// TwinCAT 3 PLC project ModbusExt_Sample
// ProgramVersion: 3.1.4026.27
// libraries:
//   ModbusExt2, * (Beckhoff Automation)
//   Tc2_SerialCom, * (Beckhoff Automation GmbH)
//   Tc2_Standard, * (Beckhoff Automation GmbH)
//   Tc2_System, * (Beckhoff Automation GmbH)
//   Tc2_Utilities, * (Beckhoff Automation GmbH)
// project tree:
//   GVLs/ GVL_IO.TcGVL, GVL_Site.TcGVL
//   / PlcTask.TcTTO
//   POUs/ MAIN.TcPOU
//   POUs/Profiles/ FB_Mb_AbbCorMeter.TcPOU, FB_Mb_DiagDemo.TcPOU, FB_Mb_FlowMeter.TcPOU, FB_Mb_TestGood.TcPOU, FB_Mb_TestValve123.TcPOU
// (motion and I/O tree: see PLC project modbusext2)
// real-time tasks:
//   TASK PlcTask1: cycle T#10ms, priority 21, ADS port 351
//   TASK PlcTask: cycle T#10ms, priority 20, ADS port 350

CONFIGURATION ModbusExt_Sample
    RESOURCE PLC ON TwinCAT3
        TASK PlcTask(INTERVAL := T#10ms, PRIORITY := 20);
        PROGRAM MAIN WITH PlcTask : MAIN;
    END_RESOURCE
END_CONFIGURATION

// ---- GVLs/GVL_IO.TcGVL
{attribute 'qualified_only'}
VAR_GLOBAL
	stEl6In1  AT %I* : EL6inData22B;
	stEl6Out1 AT %Q* : EL6outData22B;
END_VAR

// ---- GVLs/GVL_Site.TcGVL
{attribute 'qualified_only'}
VAR_GLOBAL
	{attribute 'TcInitSymbol'}
	sTcpHost   : STRING(15) := '127.0.0.1';
	{attribute 'TcInitSymbol'}
	nTcpPort   : UINT := 502;
	{attribute 'TcInitSymbol'}
	nDemoUnit  : USINT := 1;
	{attribute 'TcInitSymbol'}
	nMeterUnit : USINT := 1;
END_VAR

// ---- POUs/MAIN.TcPOU
PROGRAM MAIN
VAR
	// Transports — call before the devices that use them
	fbTcp          : FB_MbTransportTcp;
	fbRs485        : FB_MbTransportRtu;

	// Devices
	fbDemo         : FB_Mb_DiagDemo;
	fbMeter        : FB_Mb_TestGood;
	fbTemp		   : FB_ModbusDevice;

	// Write handshake example
	fSetpointCmd   : LREAL;
	bWriteSetpoint : BOOL;
END_VAR

// ---- Transports ----
fbTcp(sHost := GVL_Site.sTcpHost, nPort := GVL_Site.nTcpPort);
fbRs485(pComIn := ADR(GVL_IO.stEl6In1), pComOut := ADR(GVL_IO.stEl6Out1), nSizeComIn := SIZEOF(GVL_IO.stEl6In1));

// ---- Devices ----
fbDemo(itfTransport := fbTcp,   nUnitId := GVL_Site.nDemoUnit,  bEnable := TRUE);
fbMeter(itfTransport := fbRs485, nUnitId := GVL_Site.nMeterUnit, bEnable := TRUE, sLogName := 'FlowMeter_Inlet');

// ---- Write handshake: set fSetpointCmd, pulse bWriteSetpoint ----
IF bWriteSetpoint AND NOT fbDemo.Setpoint.bWriteReq AND NOT fbDemo.Setpoint.bWriteBusy THEN
	fbDemo.Setpoint.fWriteValue := fSetpointCmd;
	fbDemo.Setpoint.bWriteReq   := TRUE;
END_IF

IF fbDemo.Setpoint.bWriteDone OR fbDemo.Setpoint.bWriteErr THEN
	fbDemo.Setpoint.bWriteReq := FALSE;
	bWriteSetpoint            := FALSE;
END_IF

END_PROGRAM

// ---- POUs/Profiles/FB_Mb_DiagDemo.TcPOU
(*@ModbusExt.Profile v1 - managed by ModbusExt Profile Editor. One point per line.*)
FUNCTION_BLOCK FB_Mb_DiagDemo EXTENDS FB_ModbusDevice
VAR_INPUT
	Setpoint : ST_MbPoint := (nAddr := 40001);   // UInt16, read and write
	Flow     : ST_MbPoint := (nAddr := 40003, eType := E_MbType.Real32);   // 2 registers
	Temp     : ST_MbPoint := (nAddr := 40005, eType := E_MbType.Int16, fRawMin := 0, fRawMax := 1000, fEngMin := 0, fEngMax := 100, bUseFailValue := TRUE, fFailValue := -1);   // scaled, fails to -1
	Run      : ST_MbPoint := (nAddr := 1);   // coil
	Fault    : ST_MbPoint := (nAddr := 10001, ePoll := E_MbPoll.Slow);   // discrete input, slow
	Amps     : ST_MbPoint := (nAddr := 40007, eType := E_MbType.Int16);   // Test with chad and kyle, lord please work
	Volts	 : ST_MbPoint := (nAddr := 40008, eType := E_MbType.Int16);		// Test manually added from inside TC
END_VAR

Register();
SUPER^();

METHOD Register
Profile(sModel := 'DiagslaveDemo', eWordOrder := E_MbWordOrder.CDAB, tSlowPoll := T#2S);
AddPoint(Setpoint, 'Setpoint');
AddPoint(Flow, 'Flow');
AddPoint(Temp, 'Temp');
AddPoint(Run, 'Run');
AddPoint(Fault, 'Fault');
AddPoint(Amps, 'Amps');
END_METHOD

END_FUNCTION_BLOCK

// ---- POUs/Profiles/FB_Mb_TestGood.TcPOU
FUNCTION_BLOCK FB_Mb_TestGood EXTENDS FB_ModbusDevice
VAR_INPUT
	// Holding registers: 40001..40004 contiguous, 40010 within gap 8 -> one block
	Hr1    : ST_MbPoint := (nAddr := 40001);
	Hr2    : ST_MbPoint := (nAddr := 40002, eType := E_MbType.Int16, fRawMin := 0, fRawMax := 1000, fEngMin := 0, fEngMax := 100);
	Hr3    : ST_MbPoint := (nAddr := 40003, eType := E_MbType.Real32);
	Hr4    : ST_MbPoint := (nAddr := 40010, eType := E_MbType.UInt32);
	// Gap > 8 -> second block
	Hr5    : ST_MbPoint := (nAddr := 40100, eType := E_MbType.Text, nRegs := 8);
	// Slow -> its own block
	Hr6    : ST_MbPoint := (nAddr := 40116, ePoll := E_MbPoll.Slow);
	// Off -> no block
	Hr7    : ST_MbPoint := (nAddr := 40200, ePoll := E_MbPoll.Off);
	// Far away -> third fast HR block
	Hr8    : ST_MbPoint := (nAddr := 40400);
	Hr9    : ST_MbPoint := (nAddr := 40410);
	Hr10   : ST_MbPoint := (nAddr := 40420);
	Status : ST_MbPoint := (nAddr := 40300, eType := E_MbType.RegisterBit, nBit := 3);
	// Input registers, contiguous -> one block
	Ir1    : ST_MbPoint := (nAddr := 30001, eType := E_MbType.Real32);
	Ir2    : ST_MbPoint := (nAddr := 30003, eType := E_MbType.UInt32);
	// Coils and a discrete input
	Coil1  : ST_MbPoint := (nAddr := 1);
	Coil2  : ST_MbPoint := (nAddr := 2);
	Di1    : ST_MbPoint := (nAddr := 10001);
END_VAR

Register();
SUPER^();

//FB_Init is always available implicitly and it is used primarily for initialization.
//The return value is not evaluated. For a specific influence, you can also declare the
//methods explicitly and provide additional code there with the standard initialization
//code. You can evaluate the return value.
METHOD FB_Init: BOOL
VAR_INPUT
    bInitRetains: BOOL; // TRUE: the retain variables are initialized (reset warm / reset cold)
    bInCopyCode: BOOL;  // TRUE: the instance will be copied to the copy code afterward (online change)   
END_VAR
Register();
END_METHOD

METHOD FB_Reinit: BOOL
VAR_INPUT   
END_VAR
Register();
END_METHOD

METHOD PRIVATE Register
Profile(sModel := 'TestGood', eWordOrder := E_MbWordOrder.CDAB);
AddPoint(Hr1, 'Hr1');
AddPoint(Hr2, 'Hr2');
AddPoint(Hr3, 'Hr3');
AddPoint(Hr4, 'Hr4');
AddPoint(Hr5, 'Hr5');
AddPoint(Hr6, 'Hr6');
AddPoint(Hr7, 'Hr7');
AddPoint(Hr8, 'Hr8');
AddPoint(Hr9, 'Hr9');
AddPoint(Hr10, 'Hr10');
AddPoint(Status, 'Status');
AddPoint(Ir1, 'Ir1');
AddPoint(Ir2, 'Ir2');
AddPoint(Coil1, 'Coil1');
AddPoint(Coil2, 'Coil2');
AddPoint(Di1, 'Di1');
END_METHOD

END_FUNCTION_BLOCK

// ---- POUs/Profiles/FB_Mb_AbbCorMeter.TcPOU
(*@ModbusExt.Profile v1 - managed by ModbusExt Profile Editor. One point per line.*)
FUNCTION_BLOCK FB_Mb_AbbCorMeter EXTENDS FB_ModbusDevice
VAR_INPUT
	Flow     : ST_MbPoint := (nAddr := 40001, eType := E_MbType.Int16);   // replace me
	Pressure : ST_MbPoint := (nAddr := 40002, eType := E_MbType.Int16);
	Temp     : ST_MbPoint := (nAddr := 40003, eType := E_MbType.Int16, ePoll := E_MbPoll.Slow);
END_VAR

Register();
SUPER^();

METHOD PRIVATE Register
Profile(sModel := 'AbbCorMeter');
AddPoint(Flow, 'Flow');
AddPoint(Pressure, 'Pressure');
AddPoint(Temp, 'Temp');
END_METHOD

END_FUNCTION_BLOCK

// ---- POUs/Profiles/FB_Mb_FlowMeter.TcPOU
(*@ModbusExt.Profile v1 - managed by ModbusExt Profile Editor. One point per line.*)
FUNCTION_BLOCK FB_Mb_FlowMeter EXTENDS FB_ModbusDevice
VAR_INPUT
	Pressure : ST_MbPoint := (nAddr := 40001, eType := E_MbType.Int16, fRawMin := -16000, fRawMax := 16000, fEngMin := 0, fEngMax := 120);   // replace me
	Temp     : ST_MbPoint := (nAddr := 40002, eType := E_MbType.Int16, fGain := 1.8, fOffset := 32);
	Flow     : ST_MbPoint := (nAddr := 40003);
	Viscos   : ST_MbPoint := (nAddr := 40004);
END_VAR

Register();
SUPER^();

METHOD PRIVATE Register
Profile(sModel := 'FlowMeter');
AddPoint(Pressure, 'Pressure');
AddPoint(Temp, 'Temp');
AddPoint(Flow, 'Flow');
AddPoint(Viscos, 'Viscos');
END_METHOD

END_FUNCTION_BLOCK

// ---- POUs/Profiles/FB_Mb_TestValve123.TcPOU
(*@ModbusExt.Profile v1 - managed by ModbusExt Profile Editor. One point per line.*)
FUNCTION_BLOCK FB_Mb_TestValve123 EXTENDS FB_ModbusDevice
VAR_INPUT
	Point1 : ST_MbPoint := (nAddr := 40001);   // replace me
	Level  : ST_MbPoint := (nAddr := 40002, eType := E_MbType.Int16);
END_VAR

Register();
SUPER^();

METHOD PRIVATE Register
Profile(sModel := 'TestValve123');
AddPoint(Point1, 'Point1');
AddPoint(Level, 'Level');
END_METHOD

END_FUNCTION_BLOCK
